FUNCTION_BLOCK ReportScrollOffset (* Service Interface Block: reports the current scroll offset (in px) of a *_Scrolling_Content container to the ECU's VT scroll-visibility gate *)
  (* Standard: ISO 11783-6; Description: Copyright (c) 2026 Meisterschulen am Ostbahnhof This program and the accompanying materials are made available under the terms of the Eclipse Public License 2.0 which is available at https://www.eclipse.org/legal/epl-2.0/ SPDX-License-Identifier: EPL-2.0 Sits inside the ScrollFS FBNetwork, parallel to MoveList/ListY (same Ramp.INITO/Ramp.CNF triggers, same Snap.OUT.u16ListContentId/i32RowHeight sources). Multiplies i32Pos (Ramp.OUT, the current row index) by i32RowHeight and reports the resulting pixel offset to the ECU's VtMaskVisibility module (VtMaskVisibility_OnScroll(), Application/components/App_VTClient/) so row-content Q_* commands can be gated on whether their row is currently within the visible scroll window (BERICHT_2026-09-18_VT_SICHTBARKEITS_KONZEPT.md Section 4.4). Deliberately a plain, non-VT-command Basic FB (no CQ_VTCommandBase inheritance) - it does not participate in the mask-visibility notifyAllVTReady() burst mechanism, so it cannot be reentered by it. See Workspace_Scroll/SCROLL_KONZEPT.md for the scroll module this is a helper of. *)
  (* Version 1.0, 2026-09-21, Franz Höpfinger, Meisterschulen am Ostbahnhof, initial API and implementation and/or initial documentation *)
  PACKAGE isobus::UT::Q::helpers;
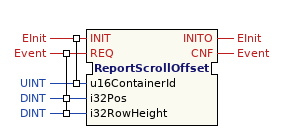
  EVENT_INPUT
    INIT : EInit WITH u16ContainerId; (* Service Initialization - latch the container ID *)
    REQ WITH i32Pos, i32RowHeight; (* Service Request - report the current position *)
  END_EVENT
  EVENT_OUTPUT
    INITO : EInit; (* Initialization Confirm *)
    CNF; (* Confirmation of Requested Service *)
  END_EVENT
  VAR_INPUT
    u16ContainerId : UINT; (* Object ID of the *_Scrolling_Content container this instance reports for - latched once at INIT *)
    i32Pos : DINT; (* Current scroll position (0..PosMax, in rows) - same value Q_ChildPosition's Y-position is derived from *)
    i32RowHeight : DINT; (* Row height in px, used to convert i32Pos into a pixel offset *)
  END_VAR
END_FUNCTION_BLOCK
